Universal Robots PolyScope program: 4exMove.urp

Program 4exMove (installation=default directory=/home/ur/ursim-current/programs createdIn=5.11.8.1010444 lastSavedIn=5.11.8.1010444 robotSerialNumber=20195399999)
Calibrated DH parameters: a=[0, -0.24355, -0.2132, 0, 0, 0]; d=[0.15185, 0, 0, 0.13105, 0.08535, 0.0921]; alpha=[1.570796, 0, 0, 1.570796, -1.570796, 0]; deltaTheta=[0, 0, 0, 0, 0, 0]
BeforeStart
  Script file /home/ur/ursim-current/programs/Script/4_Ex_Move.script
    | def Move(x, y, z, rx, ry, rz, dX, dY, dZ):
    | 	movel(p[x, y, z, rx, ry, rz], a=1, v=1)
    | 	sleep(1.0)
    | 	x = x + dX
    | 	y = y + dY
    | 	z = z + dZ
    | 	movel(p[x, y, z, rx, ry, rz], a=1, v=1)
    | 	sleep(1.0)
    | end
  'Start position'
  x := 0.0
  y := -0.2
  z := 0.3
  rx := 0
  ry := 3.14
  rz := 0
  'going to start position via movej'
  Script: movej(p[x,y,z,rx,ry,rz],a=1,v=1)
  'movement on x,y,z (mesurements in [m])'
  deltaX := 0.25
  deltaY := 0
  deltaZ := 0
Robot Program (runOnlyOnce=false)
  Wait Sleep waitTime=0.01
  Script: Move(x,y,z,rx,ry,rz,deltaX,deltaY, deltaZ)
